{attribute 'GeneratedUsingTerminal: ELX5151-0000-0016'}
{attribute addProperty BoxType "ELX5151-0000-0016"}
{attribute addProperty Id "ControlAT %Q*Control_BD9A418F1Set_counter_valueAT %Q*UINT2"}
{attribute addProperty CRC "785852399"}
{attribute addProperty Size "3"}
TYPE ENC_Control_compact_2ED727EF :
STRUCT
	{attribute addProperty Name "Control"}
	Control AT %Q* : Control_BD9A418F;
	{attribute addProperty Name "Set_counter_value"}
	Set_counter_value AT %Q* : UINT;
END_STRUCT
END_TYPE

(* stored: Version 1.2.0.0, ProductVersion 3.1.4024.9
   DUT ENC_Control_compact_2ED727EF: Id {f70bb0e7-0f09-4572-afbe-bd9869c253b1} *)
